SUBAPPLICATION SubApp_PC_A (* Geraet A (Station 11, 192.168.1.11): wie Training_11, aber Transport-Layer gebuendelt - statt je 2x AX_SUBSCRIBE_1/AX_CLIENT_1_0 (4 einzelne Netzwerk-Bausteine, 4 Konstanten) uebernimmt EIN A2X2_CLIENT_2_0_SUBSCRIBE_2 (Socket) den kompletten Roundtrip fuer UP+DOWN in je einem CLIENT_2_0/SUBSCRIBE_2 (2 Werte pro Aufruf, 2 Konstanten). Die 4 lokalen Bausteine (2 SoftKeys + 2 GreenWhiteBackground) stecken gebuendelt in MyLib::sys::Softkey2_TO_A2X2_BG, das nach aussen nur einen einzigen A2X2-Plug zeigt - dieser wird direkt in den Netzwerk-Baustein gesteckt. *)
  (* Standard: 61499-2; Description: Copyright (c) 2026 Meisterschulen am Ostbahnhof This program and the accompanying materials are made available under the terms of the Eclipse Public License 2.0 which is available at https://www.eclipse.org/legal/epl-2.0/ SPDX-License-Identifier: EPL-2.0 *)
  (* Version 1.0, 2026-09-05, Franz Höpfinger, Meisterschulen am Ostbahnhof, initial API and implementation and/or initial documentation *)
  PACKAGE subapp::Training_12_OPC_UA_RES;
  IMPORT Uebungen::const::UT::DefaultPool::SoftKey_F1;
  IMPORT Uebungen::const::UT::DefaultPool::SoftKey_F2;
  IMPORT VV::const::OPC_UA::myOpcUaAddresses::SW2_PRESS_REMOTE_WRITE;
  IMPORT VV::const::OPC_UA::myOpcUaAddresses::SW2_STATE_LOCAL_READ;
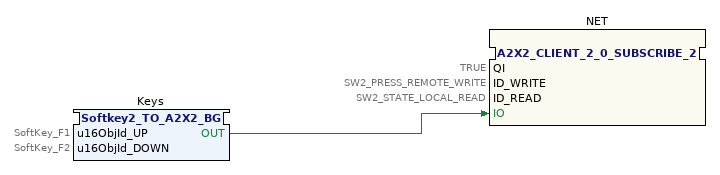
  FBS
    NET : adapter::net::A2X2_CLIENT_2_0_SUBSCRIBE_2(QI := TRUE, ID_WRITE := SW2_PRESS_REMOTE_WRITE, ID_READ := SW2_STATE_LOCAL_READ);
  END_FBS
  SUBAPPS
    Keys : MyLib::sys::Softkey2_TO_A2X2_BG(u16ObjId_UP := SoftKey_F1, u16ObjId_DOWN := SoftKey_F2);
  END_SUBAPPS
  ADAPTER_CONNECTIONS
    Keys.OUT TO NET.IO;
  END_CONNECTIONS
END_SUBAPPLICATION
